# EPICS IOC start-up script: iocsh/pace5000.iocsh
# ### pace5000 iocsh ###
# ######################
#
# P 		- Required, system level
# R		- Required, device level

dbLoadRecords("pace5000.db", "P=$(SYS), R=$(DEV), PORT=$(PORT)")
